(*
    This function block is responsible for printing the results of the assertions using the built-in
    ADSLOGSTR functionality provided by the Tc2_System library. This sends the result using ADS, which
    is consumed by the error list of Visual Studio.
*)
FUNCTION_BLOCK FB_ADSAssertMessageFormatter IMPLEMENTS I_AssertMessageFormatter

METHOD LogAssertFailure
VAR_INPUT
    Expected : STRING;
    Actual : STRING;
    Message : Tc2_System.T_MaxString;
    TestInstancePath : Tc2_System.T_MaxString;
END_VAR
VAR
    TestInstancePathCleaned : Tc2_System.T_MaxString;
    FinalMessage : Tc2_System.T_MaxString;
END_VAR
TestInstancePathCleaned := F_RemoveInstancePathAndProjectNameFromTestInstancePath(TestInstancePath);
FinalMessage := Tc2_Standard.CONCAT(STR1 := 'FAILED TEST $'', STR2 := TestInstancePathCleaned);
FinalMessage := Tc2_Standard.CONCAT(STR1 := FinalMessage, STR2 := '$'');

IF Tc2_Standard.LEN(STR := Expected) > 0 THEN
    FinalMessage := Tc2_Standard.CONCAT(STR1 := FinalMessage, STR2 := ', EXP: ');
    FinalMessage := Tc2_Standard.CONCAT(STR1 := FinalMessage, STR2 := Expected);
END_IF
IF Tc2_Standard.LEN(STR := Actual) > 0 THEN
    FinalMessage := Tc2_Standard.CONCAT(STR1 := FinalMessage, STR2 := ', ACT: ');
    FinalMessage := Tc2_Standard.CONCAT(STR1 := FinalMessage, STR2 := Actual);
END_IF
IF Tc2_Standard.LEN(STR := Message) > 0 THEN
    FinalMessage := Tc2_Standard.CONCAT(STR1 := FinalMessage, STR2 := ', MSG: %s ');
END_IF
Tc2_System.ADSLOGSTR(msgCtrlMask := Tc2_System.ADSLOG_MSGTYPE_ERROR,
                     msgFmtStr := FinalMessage,
                     strArg := Message);
END_METHOD

METHOD PUBLIC LogMessageError
VAR_INPUT
    Expected : STRING;
    Actual : STRING;
    Message : Tc2_System.T_MaxString;
    TestInstancePath : Tc2_System.T_MaxString;
END_VAR
VAR
    sTestInstancePathCleaned : Tc2_System.T_MaxString;
    sFinalMessage : Tc2_System.T_MaxString;
END_VAR
sTestInstancePathCleaned := F_RemoveInstancePathAndProjectNameFromTestInstancePath(TestInstancePath);
sFinalMessage := Tc2_Standard.CONCAT('FAILED TEST $'', sTestInstancePathCleaned);
sFinalMessage := Tc2_Standard.CONCAT(sFinalMessage, '$'');

IF Tc2_Standard.LEN(STR := Expected) > 0 THEN
    sFinalMessage := Tc2_Standard.CONCAT(sFinalMessage, ', EXP: ');
    sFinalMessage := Tc2_Standard.CONCAT(sFinalMessage, Expected);
END_IF
IF Tc2_Standard.LEN(STR := Actual) > 0 THEN
    sFinalMessage := Tc2_Standard.CONCAT(sFinalMessage, ', ACT: ');
    sFinalMessage := Tc2_Standard.CONCAT(sFinalMessage, Actual);
END_IF
IF Tc2_Standard.LEN(STR := Message) > 0 THEN
    sFinalMessage := Tc2_Standard.CONCAT(sFinalMessage, ', MSG: %s ');
END_IF
Tc2_System.ADSLOGSTR(msgCtrlMask := Tc2_System.ADSLOG_MSGTYPE_ERROR,
                     msgFmtStr := sFinalMessage,
                     strArg := Message);
END_METHOD

END_FUNCTION_BLOCK

(* stored: Version 1.1.0.1, ProductVersion 3.1.4022.12
   POU FB_ADSAssertMessageFormatter: Id {54911d7d-b4a4-43a8-a981-a2fc14a13f71}, SpecialFunc None
   Method LogAssertFailure: Id {48cbc6b0-5380-44b8-a045-57b6ad9f189d}
   Method LogMessageError: Id {bab195d7-5e96-4c3f-8266-c59551de8d0d} *)
